(* CoDeSys 2.3 export: MqttQoS.EXP *)

(* Data type in MQTT-Utils *)
TYPE MqttQoS :
(
	MQTT_QOS_AT_MOST_ONCE := 0,
	MQTT_QOS_AT_LEAST_ONCE := 1,
	MQTT_QOS_EXACTLY_ONCE := 2
);
END_TYPE
